# EPICS IOC start-up script: test/startup/st.testSimPosRestore.iocsh
epicsEnvSet("ECM_NUMAXES",   "17")
epicsEnvSet("MOTOR_PORT",    "$(SM_MOTOR_PORT=MCU1)")

epicsEnvSet("IPADDR",        "$(SM_IPADDR=127.0.0.1)")
epicsEnvSet("IPPORT",        "$(SM_IPPORT=5000)")
epicsEnvSet("ASYN_PORT",     "$(SM_ASYN_PORT=MC_CPU1)")
epicsEnvSet("SYSPFX",        "$(SM_SYSPFX=IOC:)")
epicsEnvSet("EGU",           "$(SM_EGU=mm)")
epicsEnvSet("PREC",          "$(SM_PREC=3)")

# And this reads the input of an incremental encoder terminal
# on the EtherCAT bus. Works with the simulator.
# For real terminals the adresses must be adapted

< ethercatmcController.iocsh

# Axis 10
epicsEnvSet("AXIS_NAME",    "$(SM_AXIS_NAME=m10)")
epicsEnvSet("AXIS_NO",       "$(SM_AXIS_NO=10)")
epicsEnvSet("DESC",          "$(SM_DESC=motor10)")
epicsEnvSet("AXISCONFIG",    "cfgFile=./SimPosRestore.cfg")
epicsEnvSet("ECAXISFIELDINIT", ",DVAL=10")
< ethercatmcAxis.iocsh
< ethercatmcAxisdebug.iocsh

# Axis 11
epicsEnvSet("AXIS_NAME",    "$(SM_AXIS_NAME=m11)")
epicsEnvSet("AXIS_NO",       "$(SM_AXIS_NO=11)")
epicsEnvSet("DESC",          "$(SM_DESC=motor11)")
epicsEnvSet("AXISCONFIG",    "")
epicsEnvSet("ECAXISFIELDINIT", ",DVAL=11")
< ethercatmcAxis.iocsh
< ethercatmcAxisdebug.iocsh

# Axis 12
epicsEnvSet("AXIS_NAME",    "$(SM_AXIS_NAME=m12)")
epicsEnvSet("AXIS_NO",       "$(SM_AXIS_NO=12)")
epicsEnvSet("DESC",          "$(SM_DESC=motor12)")
epicsEnvSet("AXISCONFIG",    "cfgFile=./SimPosRestore.cfg")
epicsEnvSet("ECAXISFIELDINIT", ",DVAL=12")
< ethercatmcAxis.iocsh
< ethercatmcAxisdebug.iocsh

# Axis 13
epicsEnvSet("AXIS_NAME",    "$(SM_AXIS_NAME=m13)")
epicsEnvSet("AXIS_NO",       "$(SM_AXIS_NO=13)")
epicsEnvSet("DESC",          "$(SM_DESC=motor13)")
epicsEnvSet("AXISCONFIG",    "cfgFile=./SimPosRestore.cfg")
epicsEnvSet("ECAXISFIELDINIT", ",DVAL=13")
< ethercatmcAxis.iocsh
< ethercatmcAxisdebug.iocsh

# Axis 14
epicsEnvSet("AXIS_NAME",    "$(SM_AXIS_NAME=m14)")
epicsEnvSet("AXIS_NO",       "$(SM_AXIS_NO=14)")
epicsEnvSet("DESC",          "$(SM_DESC=motor14)")
epicsEnvSet("AXISCONFIG",    "cfgFile=./SimPosRestore.cfg")
epicsEnvSet("ECAXISFIELDINIT", ",DVAL=14")
< ethercatmcAxis.iocsh
< ethercatmcAxisdebug.iocsh

# Axis 15
epicsEnvSet("AXIS_NAME",    "$(SM_AXIS_NAME=m15)")
epicsEnvSet("AXIS_NO",       "$(SM_AXIS_NO=15)")
epicsEnvSet("DESC",          "$(SM_DESC=motor15)")
epicsEnvSet("AXISCONFIG",    "cfgFile=./SimPosRestore.cfg")
epicsEnvSet("ECAXISFIELDINIT", ",DVAL=15")
< ethercatmcAxis.iocsh
< ethercatmcAxisdebug.iocsh

# Axis 16
epicsEnvSet("AXIS_NAME",    "$(SM_AXIS_NAME=m16)")
epicsEnvSet("AXIS_NO",       "$(SM_AXIS_NO=16)")
epicsEnvSet("DESC",          "$(SM_DESC=motor16)")
epicsEnvSet("AXISCONFIG",    "cfgFile=./SimPosRestore.cfg")
epicsEnvSet("ECAXISFIELDINIT", ",DVAL=16")
< ethercatmcAxis.iocsh
< ethercatmcAxisdebug.iocsh

# Axis 17
epicsEnvSet("AXIS_NAME",    "$(SM_AXIS_NAME=m17)")
epicsEnvSet("AXIS_NO",       "$(SM_AXIS_NO=17)")
epicsEnvSet("DESC",          "$(SM_DESC=motor17)")
epicsEnvSet("AXISCONFIG",    "cfgFile=./SimPosRestore.cfg")
epicsEnvSet("ECAXISFIELDINIT", ",DVAL=17")
< ethercatmcAxis.iocsh
< ethercatmcAxisdebug.iocsh
